KUKA KRL program: wkz4_ab.src, wkz4_ab.dat

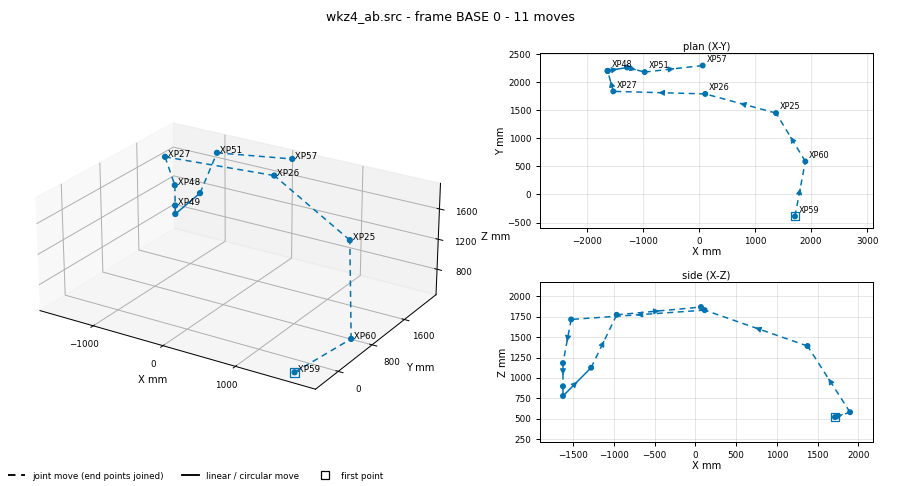
[picture p0: tool path of wkz4_ab.src in frame BASE 0, 11 of 12 moves have a stored position in this frame; points joined in program order, loops and branches not executed]
--- wkz4_ab.src ---
&ACCESS RVO2
&REL 1
&COMMENT Deposito GRIPPER ACCELO
&PARAM DISKPATH = KRC:\R1\Program
DEF wkz4_ab( )
;FOLD INI
  ;FOLD BASISTECH INI
    GLOBAL INTERRUPT DECL 3 WHEN $STOPMESS==TRUE DO IR_STOPM ( )
    INTERRUPT ON 3
    BAS (#INITMOV,0 )
  ;ENDFOLD (BASISTECH INI)
;FOLD GRIPPERTECH INI
USER_GRP(0,DUMMY,DUMMY,GDEFAULT)
;ENDFOLD (GRIPPERTECH INI)
  ;FOLD USER INI
    ;Make your modifications here

  ;ENDFOLD (USER INI)
;ENDFOLD (INI)

; Caracterização dos meios de produção:
; Changes: Deposita Gripper Accelo
; Versão Atual:11/10/2015
; Name: P13.050-R5

chk_w4_wechs_ok ( )      ; CHECK GRIPPER ACCELO

;FOLD PTP P59 CONT Vel=100 % PDAT33 Tool[1]:Gun C1 Base[0];%{PE}%R 8.2.20,%MKUKATPBASIS,%CMOVE,%VPTP,%P 1:PTP, 2:P59, 3:C_DIS, 5:100, 7:PDAT33
$BWDSTART=FALSE
PDAT_ACT=PPDAT33
FDAT_ACT=FP59
BAS(#PTP_PARAMS,100)
PTP XP59 C_DIS
;ENDFOLD
;FOLD PTP P60 CONT Vel=100 % PDAT34 Tool[1]:Gun C1 Base[0];%{PE}%R 8.2.20,%MKUKATPBASIS,%CMOVE,%VPTP,%P 1:PTP, 2:P60, 3:C_DIS, 5:100, 7:PDAT34
$BWDSTART=FALSE
PDAT_ACT=PPDAT34
FDAT_ACT=FP60
BAS(#PTP_PARAMS,100)
PTP XP60 C_DIS
;ENDFOLD

;FOLD WAIT FOR ( NOT IN 161 'DOCK 1 Deposito Ocupado' ) CONT;%{PE}%R 8.2.20,%MKUKATPBASIS,%CEXT_WAIT_FOR,%VEXT_WAIT_FOR,%P 2:, 4:NOT, 5:$IN, 6:161, 7:DOCK 1 Deposito Ocupado, 9:CONTINUE
CONTINUE
WAIT FOR  (  NOT $IN[161] )
;ENDFOLD
;FOLD WAIT FOR ( IN 219 'Posicao p/ Acoplamento OK' ) CONT;%{PE}%R 8.2.20,%MKUKATPBASIS,%CEXT_WAIT_FOR,%VEXT_WAIT_FOR,%P 2:, 4:, 5:$IN, 6:219, 7:Posicao p/ Acoplamento OK, 9:CONTINUE
CONTINUE
WAIT FOR  ( $IN[219] )
;ENDFOLD
;FOLD PULSE 167 'DOCK 1 Abrir Proteção' State=TRUE CONT Time=1 sec;%{PE}%R 8.2.20,%MKUKATPBASIS,%COUT,%VPULSE,%P 2:167, 3:DOCK 1 Abrir Proteção, 5:TRUE, 6:CONTINUE, 8:1
CONTINUE
PULSE($OUT[167], TRUE,1)
;ENDFOLD
;FOLD WAIT FOR ( IN 165 'DOCK 1 Proteção Aberta' ) CONT;%{PE}%R 8.2.20,%MKUKATPBASIS,%CEXT_WAIT_FOR,%VEXT_WAIT_FOR,%P 2:, 4:, 5:$IN, 6:165, 7:DOCK 1 Proteção Aberta, 9:CONTINUE
CONTINUE
WAIT FOR  ( $IN[165] )
;ENDFOLD
;FOLD WAIT FOR NOT ( IN 166 'DOCK 1 Proteção Fechada' ) CONT;%{PE}%R 8.2.20,%MKUKATPBASIS,%CEXT_WAIT_FOR,%VEXT_WAIT_FOR,%P 2:NOT, 4:, 5:$IN, 6:166, 7:DOCK 1 Proteção Fechada, 9:CONTINUE
CONTINUE
WAIT FOR  NOT ( $IN[166] )
;ENDFOLD
;FOLD  ;%{PE}%R 8.2.20,%MKUKATPBASIS,%CCOMMENT,%VNORMAL,%P 2:
;ENDFOLD
;FOLD PTP P25 CONT Vel=100 % PDAT14 Tool[1]:Gun C1 Base[0];%{PE}%R 8.2.20,%MKUKATPBASIS,%CMOVE,%VPTP,%P 1:PTP, 2:P25, 3:C_DIS, 5:100, 7:PDAT14
$BWDSTART=FALSE
PDAT_ACT=PPDAT14
FDAT_ACT=FP25
BAS(#PTP_PARAMS,100)
PTP XP25 C_DIS
;ENDFOLD
;FOLD PTP P26 CONT Vel=100 % PDAT15 Tool[1]:Gun C1 Base[0];%{PE}%R 8.2.20,%MKUKATPBASIS,%CMOVE,%VPTP,%P 1:PTP, 2:P26, 3:C_DIS, 5:100, 7:PDAT15
$BWDSTART=FALSE
PDAT_ACT=PPDAT15
FDAT_ACT=FP26
BAS(#PTP_PARAMS,100)
PTP XP26 C_DIS
;ENDFOLD
;FOLD PTP P27 CONT Vel=100 % PDAT28 Tool[1]:Gun C1 Base[0];%{PE}%R 8.2.20,%MKUKATPBASIS,%CMOVE,%VPTP,%P 1:PTP, 2:P27, 3:C_DIS, 5:100, 7:PDAT28
$BWDSTART=FALSE
PDAT_ACT=PPDAT28
FDAT_ACT=FP27
BAS(#PTP_PARAMS,100)
PTP XP27 C_DIS
;ENDFOLD
;FOLD PTP P48 CONT Vel=100 % PDAT30 Tool[1]:Gun C1 Base[0];%{PE}%R 8.2.20,%MKUKATPBASIS,%CMOVE,%VPTP,%P 1:PTP, 2:P48, 3:C_DIS, 5:100, 7:PDAT30
$BWDSTART=FALSE
PDAT_ACT=PPDAT30
FDAT_ACT=FP48
BAS(#PTP_PARAMS,100)
PTP XP48 C_DIS
;ENDFOLD
;FOLD PTP P49 CONT Vel=100 % PDAT31 Tool[1]:Gun C1 Base[0];%{PE}%R 8.2.20,%MKUKATPBASIS,%CMOVE,%VPTP,%P 1:PTP, 2:P49, 3:C_DIS, 5:100, 7:PDAT31
$BWDSTART=FALSE
PDAT_ACT=PPDAT31
FDAT_ACT=FP49
BAS(#PTP_PARAMS,100)
PTP XP49 C_DIS
;ENDFOLD
;FOLD ;%{PE}%R 5.4.33,%MKUKATPBASIS,%CCOMMENT,%VNORMAL,%P 2:
;ENDFOLD
;FOLD ; PONTO  DE  DEPOSITO DA  FERRAMENTA;%{PE}%R 5.4.33,%MKUKATPBASIS,%CCOMMENT,%VNORMAL,%P 2:PONTO  DE  DEPOSITO DA  FERRAMENTA
;ENDFOLD
;FOLD LIN ppegar5 Vel=0.3 m/s CPDAT13 Tool[4]:Gripper Teto Accelo Base[0];%{PE}%R 8.2.20,%MKUKATPBASIS,%CMOVE,%VLIN,%P 1:LIN, 2:ppegar5, 3:, 5:0.3, 7:CPDAT13
$BWDSTART=FALSE
LDAT_ACT=LCPDAT13
FDAT_ACT=Fppegar5
BAS(#CP_PARAMS,0.3)
LIN Xppegar5
;ENDFOLD
;FOLD  ;%{PE}%R 8.2.20,%MKUKATPBASIS,%CCOMMENT,%VNORMAL,%P 2:
;ENDFOLD
;FOLD WAIT FOR ( IN 161 'DOCK 1 Deposito Ocupado' );%{PE}%R 8.2.20,%MKUKATPBASIS,%CEXT_WAIT_FOR,%VEXT_WAIT_FOR,%P 2:, 4:, 5:$IN, 6:161, 7:DOCK 1 Deposito Ocupado, 9:
WAIT FOR  ( $IN[161] )
WAIT SEC 1
;ENDFOLD
;FOLD WAIT Time=0.3 sec;%{PE}%R 8.2.20,%MKUKATPBASIS,%CWAIT,%VWAIT,%P 3:0.3
WAIT SEC 0.3
;ENDFOLD
;FOLD OUT 224 'Bloquear MPS' State=FALSE ;%{PE}%R 8.2.20,%MKUKATPBASIS,%COUT,%VOUTX,%P 2:224, 3:Bloquear MPS, 5:FALSE, 6:
$OUT[224]=FALSE
;ENDFOLD
;FOLD OUT 223 'Desbloquear MPS' State=TRUE ;%{PE}%R 8.2.20,%MKUKATPBASIS,%COUT,%VOUTX,%P 2:223, 3:Desbloquear MPS, 5:TRUE, 6:
$OUT[223]=TRUE
;ENDFOLD
;FOLD WAIT FOR ( IN 217 'MPS Destravado' );%{PE}%R 8.2.20,%MKUKATPBASIS,%CEXT_WAIT_FOR,%VEXT_WAIT_FOR,%P 2:, 4:, 5:$IN, 6:217, 7:MPS Destravado, 9:
WAIT FOR  ( $IN[217] )
;ENDFOLD
;FOLD WAIT FOR ( NOT IN 221 'MPS Travado' );%{PE}%R 8.2.20,%MKUKATPBASIS,%CEXT_WAIT_FOR,%VEXT_WAIT_FOR,%P 2:, 4:NOT, 5:$IN, 6:221, 7:MPS Travado, 9:
WAIT FOR  (  NOT $IN[221] )
;ENDFOLD
;FOLD IBUS OFF;%{PE}%R 8.2.20,%MKUKATPBASIS,%CIBUS,%VMAP,%P 2:#OFF, 3:1
$IBUS_OFF=$IBUS_ON
$IBUS_ON=0
;ENDFOLD
;FOLD WAIT Time=0.5 sec;%{PE}%R 8.2.20,%MKUKATPBASIS,%CWAIT,%VWAIT,%P 3:0.5
WAIT SEC 0.5
;ENDFOLD

;FOLD LIN P54 Vel=0.5 m/s CPDAT33 Tool[8]:Tool Changer Base[0];%{PE}%R 8.2.20,%MKUKATPBASIS,%CMOVE,%VLIN,%P 1:LIN, 2:P54, 3:, 5:0.5, 7:CPDAT33
$BWDSTART=FALSE
LDAT_ACT=LCPDAT33
FDAT_ACT=FP54
BAS(#CP_PARAMS,0.5)
LIN XP54
;ENDFOLD

;FOLD WAIT FOR ( IN 161 'DOCK 1 Deposito Ocupado' ) CONT;%{PE}%R 8.2.20,%MKUKATPBASIS,%CEXT_WAIT_FOR,%VEXT_WAIT_FOR,%P 2:, 4:, 5:$IN, 6:161, 7:DOCK 1 Deposito Ocupado, 9:CONTINUE
CONTINUE
WAIT FOR  ( $IN[161] )
;ENDFOLD
;FOLD WAIT FOR ( NOT IN 219 'Posicao p/ Acoplamento OK' ) CONT;%{PE}%R 8.2.20,%MKUKATPBASIS,%CEXT_WAIT_FOR,%VEXT_WAIT_FOR,%P 2:, 4:NOT, 5:$IN, 6:219, 7:Posicao p/ Acoplamento OK, 9:CONTINUE
CONTINUE
WAIT FOR  (  NOT $IN[219] )
;ENDFOLD
;FOLD ;%{PE}%R 5.4.33,%MKUKATPBASIS,%CCOMMENT,%VNORMAL,%P 2:
;ENDFOLD
;FOLD PTP P51 CONT Vel=100 % PDAT23 Tool[1]:Gun C1 Base[0];%{PE}%R 8.2.20,%MKUKATPBASIS,%CMOVE,%VPTP,%P 1:PTP, 2:P51, 3:C_DIS, 5:100, 7:PDAT23
$BWDSTART=FALSE
PDAT_ACT=PPDAT23
FDAT_ACT=FP51
BAS(#PTP_PARAMS,100)
PTP XP51 C_DIS
;ENDFOLD
;FOLD PTP P57 CONT Vel=100 % PDAT29 Tool[1]:Gun C1 Base[0];%{PE}%R 8.2.20,%MKUKATPBASIS,%CMOVE,%VPTP,%P 1:PTP, 2:P57, 3:C_DIS, 5:100, 7:PDAT29
$BWDSTART=FALSE
PDAT_ACT=PPDAT29
FDAT_ACT=FP57
BAS(#PTP_PARAMS,100)
PTP XP57 C_DIS
;ENDFOLD

MBINI_2 ( )

;FOLD PTP HOME Vel=100 % DEFAULT;%{PE}%R 8.2.20,%MKUKATPBASIS,%CMOVE,%VPTP,%P 1:PTP, 2:HOME, 3:, 5:100, 7:DEFAULT
$BWDSTART=FALSE
PDAT_ACT=PDEFAULT
FDAT_ACT=FHOME
BAS(#PTP_PARAMS,100)
$H_POS=XHOME
PTP XHOME
;ENDFOLD

;FOLD PULSE 168 'DOCK 1 Fechar Proteção' State=TRUE Time=1 sec;%{PE}%R 8.2.20,%MKUKATPBASIS,%COUT,%VPULSE,%P 2:168, 3:DOCK 1 Fechar Proteção, 5:TRUE, 6:, 8:1
PULSE($OUT[168], TRUE,1)
;ENDFOLD

END

--- wkz4_ab.dat ---
&ACCESS RVO2
&REL 1
&COMMENT Deposito GRIPPER ACCELO
&PARAM DISKPATH = KRC:\R1\Program
DEFDAT wkz4_ab
;FOLD EXTERNAL DECLARATIONS;%{PE}%MKUKATPBASIS,%CEXT,%VCOMMON,%P
;FOLD GRIPPERTECH EXT
EXT  H50 (INT  :IN,INT  :IN,INT  :IN,GRP_TYP  :IN )
;ENDFOLD (GRIPPERTECH EXT)
;FOLD SPOTTECH EXT
EXT  USERSPOT (S_COMMAND  :IN,SPOT_TYPE  :IN )
;ENDFOLD (SPOTTECH EXT)
;FOLD BASISTECH EXT;%{PE}%MKUKATPBASIS,%CEXT,%VEXT,%P
EXT  BAS (BAS_COMMAND  :IN,REAL  :IN )
DECL INT SUCCESS
;ENDFOLD (BASISTECH EXT)
;FOLD USER EXT;%{E}%MKUKATPUSER,%CEXT,%VEXT,%P
;Make your modifications here

;ENDFOLD (USER EXT)
;ENDFOLD (EXTERNAL DECLARATIONS)
;# ============ START PATH : zac_p13050r5_01 =============
DECL BASIS_SUGG_T LAST_BASIS={POINT1[] "P60                     ",POINT2[] "P60                     ",CP_PARAMS[] "CPDAT33                 ",PTP_PARAMS[] "PDAT34                  ",CONT[] "C_DIS                   ",CP_VEL[] "2                       ",PTP_VEL[] "100                     ",SYNC_PARAMS[] "SYNCDAT                 ",SPL_NAME[] "S0                      "}
DECL LDAT LCPDAT13={VEL 2.0,ACC 100.0,APO_DIST 100.0,APO_FAC 50.0,AXIS_VEL 100.0,AXIS_ACC 100.0,ORI_TYP #VAR,CIRC_TYP #BASE,JERK_FAC 50.0,GEAR_JERK 50.0,EXAX_IGN 0}
DECL E6POS XPPEGAR5={X -1624.078,Y 2203.30396,Z 778.92627,A 90.5218201,B -0.364258111,C 179.962006,S 2,T 35,E1 0.0,E2 0.0,E3 0.0,E4 0.0,E5 0.0,E6 0.0}
DECL FDAT Fppegar5={TOOL_NO 4,BASE_NO 0,IPO_FRAME #BASE,POINT2[] " ",TQ_STATE FALSE}
DECL PDAT PPDAT14={VEL 100.0,ACC 100.0,APO_DIST 100.0,APO_MODE #CDIS}
DECL E6POS XP25={X 1376.67395,Y 1449.92505,Z 1392.13306,A 140.708405,B 5.35630322,C 128.090698,S 2,T 3,E1 0.0,E2 0.0,E3 0.0,E4 0.0,E5 0.0,E6 0.0}
DECL FDAT FP25={TOOL_NO 4,BASE_NO 0,IPO_FRAME #BASE,POINT2[] " ",TQ_STATE FALSE}
DECL PDAT PPDAT15={VEL 100.0,ACC 100.0,APO_DIST 100.0,APO_MODE #CDIS}
DECL E6POS XP26={X 114.384697,Y 1791.67603,Z 1832.51794,A 93.6138611,B -41.1381302,C 172.815201,S 2,T 43,E1 0.0,E2 0.0,E3 0.0,E4 0.0,E5 0.0,E6 0.0}
DECL FDAT FP26={TOOL_NO 4,BASE_NO 0,IPO_FRAME #BASE,POINT2[] " ",TQ_STATE FALSE}
DECL E6POS XP27={X -1523.85303,Y 1837.24402,Z 1718.46106,A 95.3921967,B -33.0946808,C -177.610306,S 2,T 35,E1 0.0,E2 0.0,E3 0.0,E4 0.0,E5 0.0,E6 0.0}
DECL FDAT FP27={TOOL_NO 4,BASE_NO 0,IPO_FRAME #BASE,POINT2[] " ",TQ_STATE FALSE}
DECL E6POS XP48={X -1624.32104,Y 2200.73193,Z 1182.51404,A 90.5219269,B -0.364119887,C 179.961807,S 2,T 35,E1 0.0,E2 0.0,E3 0.0,E4 0.0,E5 0.0,E6 0.0}
DECL FDAT FP48={TOOL_NO 4,BASE_NO 0,IPO_FRAME #BASE,POINT2[] " ",TQ_STATE FALSE}
DECL E6POS XP49={X -1624.14197,Y 2202.53296,Z 898.42688,A 90.5211792,B -0.3628304,C 179.960999,S 2,T 35,E1 0.0,E2 0.0,E3 0.0,E4 0.0,E5 0.0,E6 0.0}
DECL FDAT FP49={TOOL_NO 4,BASE_NO 0,IPO_FRAME #BASE,POINT2[] " ",TQ_STATE FALSE}
DECL E6POS XP51={X -964.794922,Y 2181.07202,Z 1775.16797,A -129.070999,B 34.6863098,C 131.582001,S 2,T 43,E1 0.0,E2 0.0,E3 0.0,E4 0.0,E5 0.0,E6 0.0}
DECL FDAT FP51={TOOL_NO 8,BASE_NO 0,IPO_FRAME #BASE,POINT2[] " ",TQ_STATE FALSE}
DECL PDAT PPDAT23={VEL 100.0,ACC 100.0,APO_DIST 100.0,APO_MODE #CDIS}
DECL E6POS XP54={X -1278.76599,Y 2262.90503,Z 1126.104,A -164.479294,B 0.131105602,C 179.658203,S 2,T 35,E1 0.0,E2 0.0,E3 0.0,E4 0.0,E5 0.0,E6 0.0}
DECL FDAT FP54={TOOL_NO 8,BASE_NO 0,IPO_FRAME #BASE,POINT2[] " ",TQ_STATE FALSE}
DECL LDAT LCPDAT33={VEL 2.0,ACC 100.0,APO_DIST 100.0,APO_FAC 50.0,AXIS_VEL 100.0,AXIS_ACC 100.0,ORI_TYP #VAR,CIRC_TYP #BASE,JERK_FAC 50.0,GEAR_JERK 50.0,EXAX_IGN 0}
DECL PDAT PPDAT28={VEL 100.0,ACC 100.0,APO_DIST 100.0,APO_MODE #CDIS}
DECL E6POS XP57={X 68.7766724,Y 2297.68311,Z 1870.41895,A -20.5327492,B 37.7427597,C -119.328697,S 2,T 11,E1 0.0,E2 0.0,E3 0.0,E4 0.0,E5 0.0,E6 0.0}
DECL FDAT FP57={TOOL_NO 8,BASE_NO 0,IPO_FRAME #BASE,POINT2[] " ",TQ_STATE FALSE}
DECL PDAT PPDAT29={VEL 100.0,ACC 100.0,APO_DIST 100.0,APO_MODE #CDIS}
DECL PDAT PPDAT30={VEL 100.0,ACC 100.0,APO_DIST 100.0,APO_MODE #CDIS}
DECL PDAT PPDAT31={VEL 100.0,ACC 100.0,APO_DIST 100.0,APO_MODE #CDIS}
DECL E6POS XP59={X 1713.74902,Y -390.089294,Z 519.985718,A 179.449097,B -44.0414505,C -179.216599,S 2,T 2,E1 0.0,E2 0.0,E3 0.0,E4 0.0,E5 0.0,E6 0.0}
DECL FDAT FP59={TOOL_NO 4,BASE_NO 0,IPO_FRAME #BASE,POINT2[] " ",TQ_STATE FALSE}
DECL PDAT PPDAT33={VEL 100.0,ACC 100.0,APO_DIST 0.0,APO_MODE #CDIS}
DECL E6POS XP60={X 1898.23999,Y 588.316528,Z 579.823975,A -75.0753632,B -0.567493677,C 10.4471998,S 2,T 3,E1 0.0,E2 0.0,E3 0.0,E4 0.0,E5 0.0,E6 0.0}
DECL FDAT FP60={TOOL_NO 1,BASE_NO 0,IPO_FRAME #BASE,POINT2[] " ",TQ_STATE FALSE}
DECL PDAT PPDAT34={VEL 100.0,ACC 100.0,APO_DIST 100.0,APO_MODE #CDIS}
ENDDAT
